# EPICS substitutions: sampleApp/Db/iocAdmin.substitutions
#==============================================================================
#
# Abs:  IOC Administration Records
#
# Name: iocAdmin.substitutions
#
#==============================================================================
#
# use one of
# file iocHard.db
# file iocSoft.db

file iocSoft.db
{
	{ IOC	= $(IOC)  }
}
